{attribute 'GeneratedUsingTerminal: EJ7211-9414-0030'}
{attribute addProperty BoxType "EJ7211-9414-0030"}
{attribute addProperty Id "AdsAddrAT %I*.TcoAmsAddr0DcOutputShiftAT %I*DINT4DcInputShiftAT %I*DINT4Chn0AT %I*USINT1Chn1AT %I*USINT1Chn2AT %I*USINT1StateAT %I*UINT2"}
{attribute addProperty CRC "1961062636"}
{attribute addProperty Size "13"}
TYPE InfoData_74E370EC :
STRUCT
	{attribute addProperty Name "AdsAddr"}
	AdsAddr AT %I* : .TcoAmsAddr;
	{attribute addProperty Name "DcOutputShift"}
	DcOutputShift AT %I* : DINT;
	{attribute addProperty Name "DcInputShift"}
	DcInputShift AT %I* : DINT;
	{attribute addProperty Name "Chn0"}
	Chn0 AT %I* : USINT;
	{attribute addProperty Name "Chn1"}
	Chn1 AT %I* : USINT;
	{attribute addProperty Name "Chn2"}
	Chn2 AT %I* : USINT;
	{attribute addProperty Name "State"}
	State AT %I* : UINT;
END_STRUCT
END_TYPE

(* stored: Version 1.2.0.0, ProductVersion 3.1.4024.9
   DUT InfoData_74E370EC: Id {01e35241-46e1-41fa-be0a-27d9cf25740d} *)
